FUNCTION_BLOCK FB_ValveBase
VAR_INPUT
END_VAR
VAR_OUTPUT
END_VAR
VAR
	// For logging
    fbLogger : FB_LogMessage := (eSubsystem:=E_SubSystem.VACUUM);
   // ePrevState : E_ValvePositionState;
    tErrorPresent : R_TRIG;
    tAction : R_TRIG; // Primary action of this device (OPN_DO, etc.)
    tOverrideActivated : R_TRIG;
END_VAR

ACTION ACT_Logger:

END_ACTION

END_FUNCTION_BLOCK

(* stored: Version 1.1.0.1, ProductVersion 3.1.4024.3
   POU FB_ValveBase: Id {d216fd72-6969-4ab7-a5bc-556a1c976071}, SpecialFunc None
   Action ACT_Logger: Id {a287235d-78df-4063-a496-ba56a271188f} *)
